// TwinCAT 3 PLC project Calculator
// ProgramVersion: 3.1.4023.0
// libraries:
//   Tc2_Standard, * (Beckhoff Automation GmbH)
//   Tc2_System, * (Beckhoff Automation GmbH)
//   Tc3_Module, * (Beckhoff Automation GmbH)
//   VisuDialogs, * (System)
//   VisuSymbols,3.5.10.0,System
// project tree:
//   / GlobalTextList.TcGTLO, PlcTask.TcTTO, Visualization Manager.TcVMO (not stored)
//   POUs/ MAIN.TcPOU
//   VISUs/ Visualization.TcVIS

CONFIGURATION Calculator
    RESOURCE PLC ON TwinCAT3
        TASK PlcTask(INTERVAL := T#10ms, PRIORITY := 20);
        PROGRAM MAIN WITH PlcTask : MAIN;
    END_RESOURCE
END_CONFIGURATION

// ---- POUs/MAIN.TcPOU
PROGRAM MAIN
VAR CONSTANT
	Years:							INT := 33;
END_VAR
VAR
	FlatPrice:						REAL := 100000;
	BrokerageCommissionPercent:		REAL := 2.975;
	RealEstateTransferTaxPercent:	REAL := 3.5;
	NotaryFeesPercent:				REAL := 1.5;
	LandRegisterEntryPercent:		REAL := 0.5;
	AdditionalCostsPercent:			REAL;
	
	BrokerageCommission:			REAL;		//Maklerprovision
	RealEstateTransferTax:			REAL;		//Grunderwerbssteuer
	NotaryFees:						REAL;		//Notarkosten
	LandRegisterEntry:				REAL;		//Grundbucheintrag
	AdditionalCosts:				REAL;		//Nebenkosten
	
	FlatGrossPrice:					REAL;
	
	(* Settlement: *)
	Capital:						REAL := 20000;
	Salary:							REAL := 2000;
	CapitalPercent:					REAL;
	Credit:							REAL;
	CreditPercent:					REAL;
	MonthlyInstallment:				REAL := 500;
	SpecialInstallment:				REAL := 0;
	InterestRate:					REAL := 1.5;
	
	(* Statistics *)
	InterestAmount:					ARRAY[1..Years*12] OF REAL;
	PaidInterest:					REAL;
	PaidInterest10years:			REAL;
	RestAmount:						ARRAY[1..Years*12] OF REAL;
	PaymentYears:					INT;
	PaymentMonths:					INT;
	MoneyLoss:						REAL;
	MoneyLossMonthly:				REAL;
	i:								INT := 1;
	j:								int;
	
	(* VISU *)
	arVisu:							ARRAY[1..2] OF ARRAY[1..Years*12] OF REAL;
	arVisu2:						ARRAY[1..3] OF ARRAY[1..Years] OF REAL;
END_VAR

// Initial Conditions:
i:=									1;
MEMSET(ADR(RestAmount), 0, SIZEOF(RestAmount));
MEMSET(ADR(InterestAmount), 0, SIZEOF(InterestAmount));
MEMSET(ADR(arVisu), 0, SIZEOF(arVisu));
MEMSET(ADR(arVisu2), 0, SIZEOF(arVisu2));

// Calculations:
BrokerageCommission:=				BrokerageCommissionPercent * FlatPrice / 100;
RealEstateTransferTax:=				RealEstateTransferTaxPercent * FlatPrice / 100;
NotaryFees:=						NotaryFeesPercent * FlatPrice / 100;
LandRegisterEntry:=					LandRegisterEntryPercent * FlatPrice / 100;
AdditionalCostsPercent:=			BrokerageCommissionPercent + RealEstateTransferTaxPercent + NotaryFeesPercent + LandRegisterEntryPercent;
AdditionalCosts:=					BrokerageCommission + RealEstateTransferTax + NotaryFees + LandRegisterEntry;

FlatGrossPrice:=					AdditionalCosts + FlatPrice;
CapitalPercent:=					Capital / FlatGrossPrice * 100;
Credit:=							FlatGrossPrice - Capital;
IF Credit < 0 THEN
	Credit :=						0;
END_IF
IF Salary > 0 THEN
	CreditPercent:=					Credit / Salary;
ELSE
	CreditPercent:=					0;
END_IF

InterestAmount[i]:=					Credit * InterestRate / 100 / 12;
PaidInterest:=						InterestAmount[i];
PaidInterest10years:=				InterestAmount[i];
RestAmount[i]:=						Credit + InterestAmount[i] - MonthlyInstallment;
IF RestAmount[i] < 0 THEN
	RestAmount[i]:=				0;
END_IF
	
WHILE RestAmount[i] > 0 DO
	i:=								i + 1;
	InterestAmount[i]:=				RestAmount[i-1] * InterestRate / 100 / 12;
	PaidInterest:=					PaidInterest + InterestAmount[i];
	IF i = 120 THEN
		PaidInterest10years:=		PaidInterest;
	END_IF
	RestAmount[i] :=				RestAmount[i-1] + InterestAmount[i] - MonthlyInstallment;
	IF (i MOD 12 = 0) THEN
		RestAmount[i] :=			RestAmount[i] - SpecialInstallment;
	END_IF
	IF RestAmount[i] < 0 THEN
		RestAmount[i]:=				0;
		IF i < 120 THEN
			PaidInterest10years:=	PaidInterest;
		END_IF
	END_IF
	IF i = Years*12 THEN
		EXIT;
	END_IF
END_WHILE
MoneyLoss:=							AdditionalCosts + PaidInterest;
MoneyLossMonthly:=					MoneyLoss / i;
PaymentYears:=						i / 12;
PaymentMonths:=						i MOD 12;

(* VISU *)
FOR i := 1 TO Years*12 DO
	arVisu[1][i]:=					DINT_TO_REAL(TRUNC(InterestAmount[i]));
	arVisu[2][i]:=					DINT_TO_REAL(TRUNC(RestAmount[i]));
END_FOR
FOR i := 1 TO PaymentYears + BOOL_TO_INT(PaymentMonths > 0) DO
	arVisu2[1][i]:=					0;
	FOR j := 1 TO 12 DO
		arVisu2[1][i]:=				arVisu2[1][i] + InterestAmount[j+12*(i-1)];
	END_FOR
	arVisu2[1][i]:=					DINT_TO_REAL(TRUNC(arVisu2[1][i]));							// Paid interst
	arVisu2[2][i]:=					DINT_TO_REAL(TRUNC(RestAmount[12*i]));						// Rest credit
	arVisu2[3][i]:=					((MonthlyInstallment * 12) - arVisu2[1][i]) / Credit * 100;	// Amortization
END_FOR

END_PROGRAM

// ---- GlobalTextList.TcGTLO
TEXTLIST GlobalTextList
  599 = '%'
  988 = '%1.2f'
  93 = '%1.3f'
  775 = '%2.0'
  271 = '%2.0f'
  136 = '%3.2f'
  836 = '%4.0f'
  994 = '%4.2f'
  263 = '%5.0f'
  211 = '%5.2f'
  981 = '%6.0f'
  800 = '%7.0f'
  610 = '%f'
  48 = '%S'
  510 = 'Additional Costs % (Grunderwerbssteuer %):'
  421 = 'Additional Costs % (Nebenkosten %):'
  574 = 'Additional Costs (Nebenkosten):'
  711 = 'Amortization (%)'
  26 = 'Brokerage Commission % (Maklerprovision %):'
  152 = 'Brokerage Commission (Maklerprovision):'
  458 = 'Credit ()'
  744 = 'Credit (Kredit):'
  150 = 'Credit (Kreditl):'
  373 = 'Equity Capital (Eigenkapital):'
  6 = 'Fach'
  202 = 'Flat Gross Price (Wohnung Gesamtpreis):'
  122 = 'Flat Price'
  743 = 'Flat Price (Wohnung Gesamtpreis):'
  900 = 'Flat Price (Wohnung Preis):'
  484 = 'Interest'
  39 = 'Interest (bezahlte Zinsen):'
  954 = 'Interest (€)'
  910 = 'Interest in 10 years (bezahlte Zinsen in 10 Jahre):'
  97 = 'Interest Rate (Zinsen):'
  734 = 'Interest €'
  801 = 'Interest-10 years (bezahlte Zinsen-10 Jahre):'
  323 = 'Land Register Entry % (Grundbucheintrag %):'
  290 = 'Land Register Entry % (Grunderwerbssteuer %):'
  653 = 'Land Register Entry (Grundbucheintrag):'
  471 = 'Monate'
  628 = 'Money Loss (Geldverlust)'
  196 = 'Money Loss (Geldverlust):'
  707 = 'Money Loss Monthly (Geldverlust monatlich):'
  998 = 'Money Loss Monthly (Geldverlust):'
  434 = 'Monthly Installment (Monatesrate):'
  388 = 'Monthly Settlement (Eigenkapital):'
  356 = 'Months'
  47 = 'Months (Monate)'
  632 = 'Months (Monate):'
  621 = 'Mortgage (Hypothek)'
  215 = 'Mortgage (Hypothek):'
  583 = 'Notary Fees % (Grunderwerbssteuer %):'
  724 = 'Notary Fees % (Notarkosten %):'
  145 = 'Notary Fees (Notarkosten):'
  696 = 'Real Estate Transfer Tax % (Grunderwerbssteuer %):'
  846 = 'Real Estate Transfer Tax % (Maklerprovision %):'
  559 = 'Real Estate Transfer Tax (Grunderwerbssteuer):'
  15 = 'Rest Amount (€)'
  989 = 'Rest Amount €'
  699 = 'Salary (Gehalt) | Credit/Salary (Kredit/Gehalt):'
  824 = 'Salary (Gehalt) | Credit/Salary:'
  293 = 'Salary (Gehalt) — Credit/Salary:'
  777 = 'Salery (Gehalt) — Credit/Salery:'
  664 = 'Salery (Gehalt):'
  611 = 'Special Installment (Sondertilgung):'
  864 = 'Special Payment (Sondertilgung):'
  805 = 'Summary (Zusammenfassung)'
  123 = 'Summary (Zussamenfassung)'
  534 = 'Years (Jahre)'
  986 = 'Years (Jahre):'
  950 = '€'
END_TEXTLIST

// ---- VISUs/Visualization.TcVIS
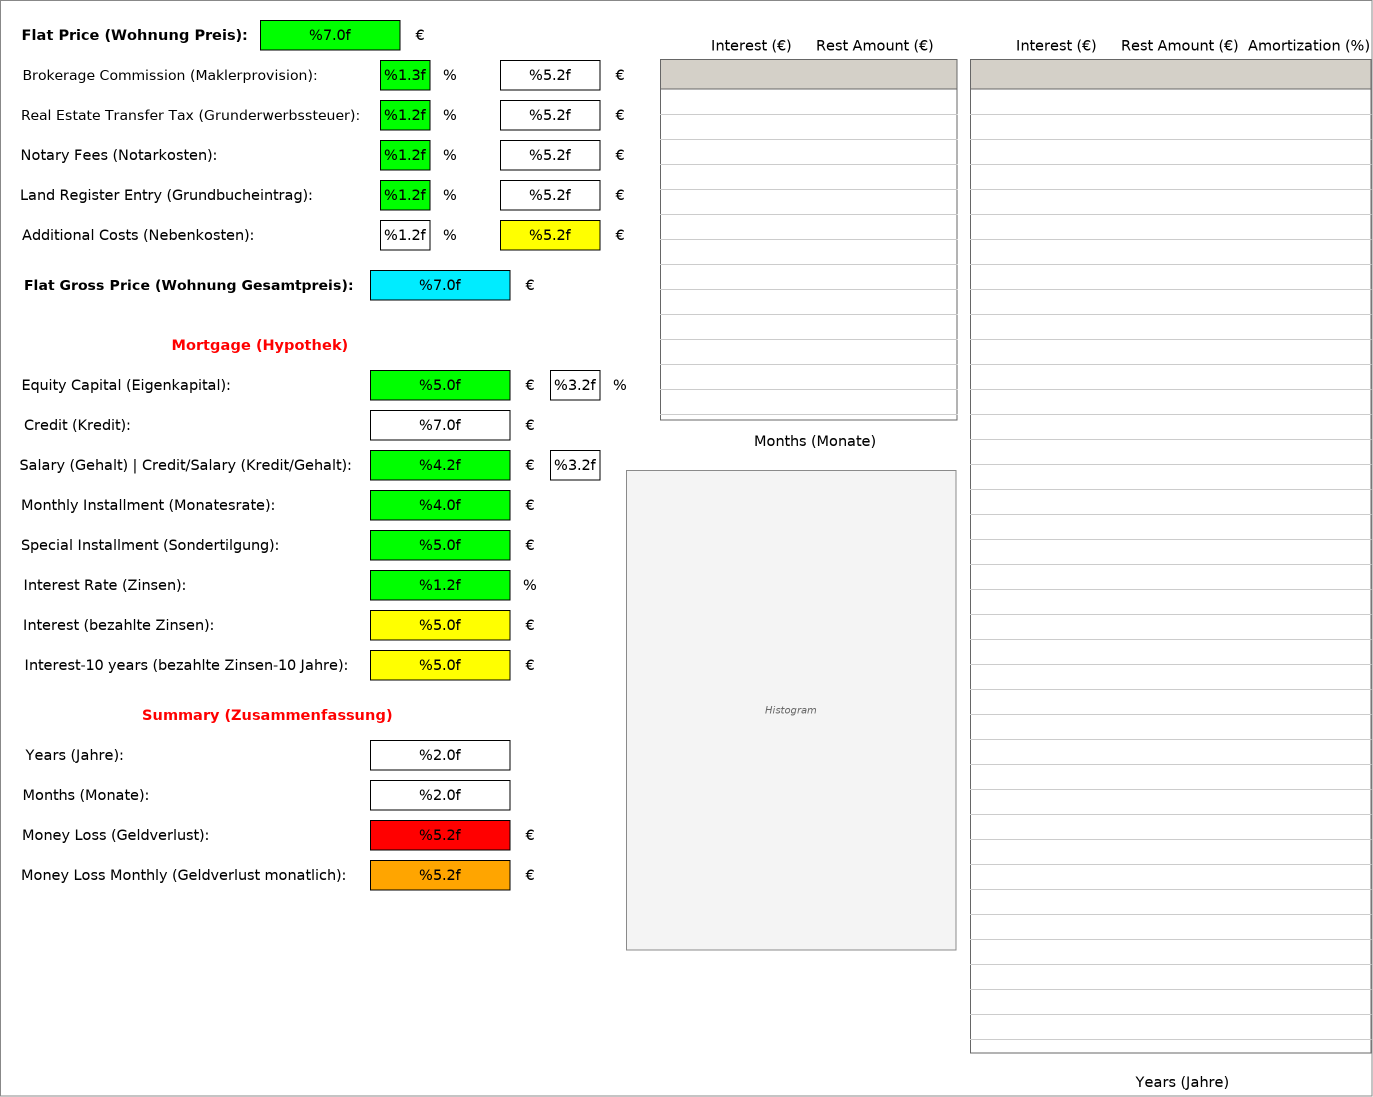
VISUALIZATION Visualization  // 1373x1097
    Textfield (20,20 230x30), "Flat Price (Wohnung Preis):"
    Rectangle (260,20 140x30), "%7.0f", text variable: MAIN.FlatPrice
        OnMouseClick: write the text variable via VisuDialogs.Numpad, min 0, max 1000000
    Rectangle (380,60 50x30), "%1.3f", text variable: MAIN.BrokerageCommissionPercent
        OnMouseClick: write the text variable via VisuDialogs.Numpad, min 0, max 10
    Rectangle (380,100 50x30), "%1.2f", text variable: MAIN.RealEstateTransferTaxPercent
        OnMouseClick: write the text variable via VisuDialogs.Numpad, min 0, max 10
    Rectangle (380,140 50x30), "%1.2f", text variable: MAIN.NotaryFeesPercent
        OnMouseClick: write the text variable via VisuDialogs.Numpad, min 0, max 10
    Rectangle (380,180 50x30), "%1.2f", text variable: MAIN.LandRegisterEntryPercent
        OnMouseClick: write the text variable via VisuDialogs.Numpad, min 0, max 10
    Rectangle (380,220 50x30), "%1.2f", text variable: MAIN.AdditionalCostsPercent
    Textfield (20,60 300x30), "Brokerage Commission (Maklerprovision):"
    Rectangle (500,60 100x30), "%5.2f", text variable: MAIN.BrokerageCommission
    Textfield (20,100 341x30), "Real Estate Transfer Tax (Grunderwerbssteuer):"
    Rectangle (500,100 100x30), "%5.2f", text variable: MAIN.RealEstateTransferTax
    Textfield (20,140 198x30), "Notary Fees (Notarkosten):"
    Rectangle (500,140 100x30), "%5.2f", text variable: MAIN.NotaryFees
    Textfield (20,180 293x30), "Land Register Entry (Grundbucheintrag):"
    Rectangle (500,180 100x30), "%5.2f", text variable: MAIN.LandRegisterEntry
    Textfield (20,220 237x30), "Additional Costs (Nebenkosten):"
    Rectangle (500,220 100x30), "%5.2f", text variable: MAIN.AdditionalCosts
    Textfield (440,60 20x30), "%"
    Textfield (440,100 20x30), "%"
    Textfield (440,140 20x30), "%"
    Textfield (440,180 20x30), "%"
    Textfield (440,220 20x30), "%"
    Textfield (610,60 20x30), "€"
    Textfield (610,100 20x30), "€"
    Textfield (610,140 20x30), "€"
    Textfield (610,180 20x30), "€"
    Textfield (610,220 20x30), "€"
    Textfield (410,20 20x30), "€"
    Textfield (20,270 338x30), "Flat Gross Price (Wohnung Gesamtpreis):"
    Rectangle (370,270 140x30), "%7.0f", text variable: MAIN.FlatGrossPrice
    Textfield (520,270 20x30), "€"
    Textfield (160,330 200x30), "Mortgage (Hypothek)"
    Textfield (20,370 213x30), "Equity Capital (Eigenkapital):"
    Rectangle (370,370 140x30), "%5.0f", text variable: MAIN.Capital
        OnMouseClick: write the text variable via VisuDialogs.Numpad, min 0, max 300000
    Textfield (520,370 20x30), "€"
    Textfield (20,410 115x30), "Credit (Kredit):"
    Rectangle (370,410 140x30), "%7.0f", text variable: MAIN.Credit
    Textfield (520,410 20x30), "€"
    Textfield (20,490 257x30), "Monthly Installment (Monatesrate):"
    Rectangle (370,490 140x30), "%4.0f", text variable: MAIN.MonthlyInstallment
        OnMouseClick: write the text variable via VisuDialogs.Numpad, min 0, max 10000
    Textfield (520,490 20x30), "€"
    Textfield (20,570 170x30), "Interest Rate (Zinsen):"
    Rectangle (370,570 140x30), "%1.2f", text variable: MAIN.InterestRate
        OnMouseClick: write the text variable via VisuDialogs.Numpad, min 0, max 5
    Textfield (520,570 20x30), "%"
    Table (660,59 297x361), data array: MAIN.arVisu
        p3854506369: MAIN.arVisu[1][INDEX]
        p1892666644: MAIN.arVisu[2][INDEX]
    Textfield (20,610 198x30), "Interest (bezahlte Zinsen):"
    Rectangle (370,610 140x30), "%5.0f", text variable: MAIN.PaidInterest
    Textfield (520,610 20x30), "€"
    Table (970,59 401x994), data array: MAIN.arVisu2
        p3854506369: MAIN.arVisu2[1][INDEX]
        p1892666644: MAIN.arVisu2[2][INDEX]
        p338671338: MAIN.arVisu2[3][INDEX]
    Textfield (20,740 110x30), "Years (Jahre):"
    Rectangle (370,740 140x30), "%2.0f", text variable: MAIN.PaymentYears
    Textfield (18,780 136x30), "Months (Monate):"
    Rectangle (370,780 140x30), "%2.0f", text variable: MAIN.PaymentMonths
    Textfield (750,426 130x30), "Months (Monate)"
    Textfield (1135,1067 95x30), "Years (Jahre)"
    Textfield (710,33 83x25), "Interest (€)"
    Textfield (815,33 120x25), "Rest Amount (€)"
    Textfield (1015,33 83x25), "Interest (€)"
    Textfield (1120,33 120x25), "Rest Amount (€)"
    Textfield (140,700 255x30), "Summary (Zusammenfassung)"
    Textfield (20,820 192x30), "Money Loss (Geldverlust):"
    Rectangle (370,820 140x30), "%5.2f", text variable: MAIN.MoneyLoss
    Textfield (520,820 20x30), "€"
    Rectangle (550,370 50x30), "%3.2f", text variable: MAIN.CapitalPercent
    Textfield (610,370 20x30), "%"
    Textfield (20,860 328x30), "Money Loss Monthly (Geldverlust monatlich):"
    Rectangle (370,860 140x30), "%5.2f", text variable: MAIN.MoneyLossMonthly
    Textfield (520,860 20x30), "€"
    Textfield (20,650 333x30), "Interest-10 years (bezahlte Zinsen-10 Jahre):"
    Rectangle (370,650 140x30), "%5.0f", text variable: MAIN.PaidInterest10years
    Textfield (520,650 20x30), "€"
    Textfield (20,450 332x30), "Salary (Gehalt) | Credit/Salary (Kredit/Gehalt):"
    Rectangle (370,450 140x30), "%4.2f", text variable: MAIN.Salary
        OnMouseClick: write the text variable via VisuDialogs.Numpad, min 0, max 150000
    Textfield (520,450 20x30), "€"
    Rectangle (550,450 50x30), "%3.2f", text variable: MAIN.CreditPercent
    Textfield (1245,33 128x25), "Amortization (%)"
    Textfield (20,530 261x30), "Special Installment (Sondertilgung):"
    Rectangle (370,530 140x30), "%5.0f", text variable: MAIN.SpecialInstallment
        OnMouseClick: write the text variable via VisuDialogs.Numpad, min 0, max 25000
    Textfield (520,530 20x30), "€"
    Histogram (626,470 330x480), scale format: %.1f, scale 0..600000
        p1518820177: MAIN.arVisu[2]
        p102497268: MAIN.arVisu[2]
        p788070771: ARRAY [1..(Years * 12)] OF REAL
END_VISUALIZATION
